FUNCTION_BLOCK AI_AX_SEL_AI (* binary selection *)
  (* Standard: 61499-2; Description: Copyright (c) 2026 HR Agrartechnik GmbH This program and the accompanying materials are made available under the terms of the Eclipse Public License 2.0 which is available at https://www.eclipse.org/legal/epl-2.0/ SPDX-License-Identifier: EPL-2.0 *)
  (* Version 1.0, 2026-04-19, Franz Höpfinger, HR Agrartechnik GmbH, initial API and implementation *)
  PACKAGE adapter::iec61131::selection;
  IMPORT eclipse4diac::core::TypeHash;
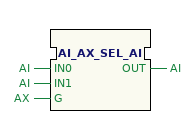
  SOCKETS
    IN0 : adapter::types::unidirectional::AI; (* Selectable input variable *)
    IN1 : adapter::types::unidirectional::AI; (* Selectable input variable *)
    G : adapter::types::unidirectional::AX; (* Selector *)
  END_SOCKETS
  PLUGS
    OUT : adapter::types::unidirectional::AI; (* Selected Output *)
  END_PLUGS
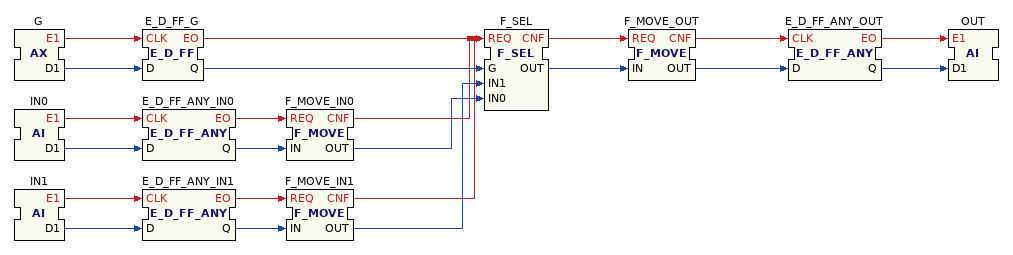
  FBS
    F_SEL : iec61131::selection::F_SEL;
    E_D_FF_ANY_OUT : iec61499::events::E_D_FF_ANY;
    F_MOVE_OUT : iec61131::selection::F_MOVE; {SET_ATTRIBUTE(DataType, INT)}
    E_D_FF_ANY_IN1 : iec61499::events::E_D_FF_ANY;
    E_D_FF_ANY_IN0 : iec61499::events::E_D_FF_ANY;
    E_D_FF_G : iec61499::events::E_D_FF;
    F_MOVE_IN0 : iec61131::selection::F_MOVE; {SET_ATTRIBUTE(DataType, INT)}
    F_MOVE_IN1 : iec61131::selection::F_MOVE; {SET_ATTRIBUTE(DataType, INT)}
  END_FBS
  EVENT_CONNECTIONS
    E_D_FF_ANY_OUT.EO TO OUT.E1;
    F_MOVE_OUT.CNF TO E_D_FF_ANY_OUT.CLK;
    F_SEL.CNF TO F_MOVE_OUT.REQ;
    G.E1 TO E_D_FF_G.CLK;
    IN0.E1 TO E_D_FF_ANY_IN0.CLK;
    IN1.E1 TO E_D_FF_ANY_IN1.CLK;
    E_D_FF_G.EO TO F_SEL.REQ;
    E_D_FF_ANY_IN0.EO TO F_MOVE_IN0.REQ;
    E_D_FF_ANY_IN1.EO TO F_MOVE_IN1.REQ;
    F_MOVE_IN1.CNF TO F_SEL.REQ;
    F_MOVE_IN0.CNF TO F_SEL.REQ;
  END_CONNECTIONS
  DATA_CONNECTIONS
    E_D_FF_ANY_OUT.Q TO OUT.D1;
    F_MOVE_OUT.OUT TO E_D_FF_ANY_OUT.D;
    F_SEL.OUT TO F_MOVE_OUT.IN;
    G.D1 TO E_D_FF_G.D;
    IN0.D1 TO E_D_FF_ANY_IN0.D;
    IN1.D1 TO E_D_FF_ANY_IN1.D;
    E_D_FF_G.Q TO F_SEL.G;
    E_D_FF_ANY_IN0.Q TO F_MOVE_IN0.IN;
    E_D_FF_ANY_IN1.Q TO F_MOVE_IN1.IN;
    F_MOVE_IN1.OUT TO F_SEL.IN1;
    F_MOVE_IN0.OUT TO F_SEL.IN0;
  END_CONNECTIONS
END_FUNCTION_BLOCK
